(* IEC 61131-3 sources: Industry-PLC-LLM/data/PLCBEAD_repo/PLCBEAD_PLCEmbed-main/PLC-BEAD/Source/GEB/DWORD_TO_DATE, 1 file *)

(* ---- DWORD_TO_DATE.ST ---- *)
FUNCTION DWORD_TO_DATE2:UDINT
	VAR_INPUT
		IN :	DWORD;
	END_VAR
	DWORD_TO_DATE2 := DWORD_TO_UDINT(IN);
END_FUNCTION

PROGRAM program0
  VAR
    LocalVar0 : DWORD;
	LocalOUT  : UDINT;
  END_VAR
  	LocalOUT := DWORD_TO_DATE2(LocalVar0);
END_PROGRAM
